TYPE DrillingComSubscribe :
STRUCT
  Request : DrillingComRequest; // contains booleans that are used to start a specific sequence.
  Equipment : DrillingComSubscribeEquipment;  // structs for equipment objects which are used by the bridges
END_STRUCT
END_TYPE

(* stored: Version 1.1.0.1
   DUT DrillingComSubscribe: Id {eba895a9-04cf-4a2f-ac8e-aca54073d0e2} *)
